// TwinCAT 3 PLC project Assembler
// ProgramVersion: 3.1.4023.0
// libraries:
//   Tc2_Standard, * (Beckhoff Automation GmbH)
//   Tc2_System, * (Beckhoff Automation GmbH)
//   Tc3_Module, * (Beckhoff Automation GmbH)
// project tree:
//   / GlobalTextList.TcGTLO, PlcTask.TcTTO, Visualization Manager.TcVMO (not stored)
//   POUs/ FB_Axxe.TcPOU, FB_Holder.TcPOU, FB_Nagel.TcPOU, FB_Robot.TcPOU, FB_Schraubendreher.TcPOU, MAIN.TcPOU, Mashine.TcPOU, Sensore.TcPOU
//   VISUs/ Visualization.TcVIS

CONFIGURATION Assembler
    RESOURCE PLC ON TwinCAT3
        TASK PlcTask(INTERVAL := T#10ms, PRIORITY := 20);
        PROGRAM MAIN WITH PlcTask : MAIN;
    END_RESOURCE
END_CONFIGURATION

// ---- POUs/MAIN.TcPOU
PROGRAM MAIN
VAR
	Position1:INT;
	Position2:INT;
	Position3:INT;
	MyMashine:Mashine;
END_VAR

MyMashine();

END_PROGRAM

// ---- POUs/Mashine.TcPOU
FUNCTION_BLOCK Mashine
VAR_INPUT
END_VAR
VAR_OUTPUT
END_VAR
VAR
	DelayTimer:TON;
	MyRobot:FB_Robot;
	l_Schraubendreher1:FB_Schraubendreher;
	l_Schraubendreher2:FB_Schraubendreher;
	l_i_Step_Stat:INT;
	l_i_Model1:INT:=0;
	l_i_Model2:INT:=0;
	l_i_Model3:INT:=0;
	l_i_Move_Step_Stat:INT;
	Holder:ARRAY[1..11] OF FB_Holder;
	Nagel:ARRAY[1..11] OF FB_Nagel;
	RoboCurrent:UINT:=1;
	Dre1Current:UINT:=1;
	Dre2Current:UINT:=1;
	DoneCurrent:uINT:=1;
	Sensore1:Sensore;
	Sensore2:Sensore;
	Sensore3:Sensore;
END_VAR

MyRobot.i_HOZAxxe.M_SetAxxeValues(AxxeMinPos:=0,AxxeMaxPos:=50);
MyRobot.i_GRFLeftAxxe.M_SetAxxeValues(AxxeMinPos:=0,AxxeMaxPos:=2);
MyRobot.i_GRFRightAxxe.M_SetAxxeValues(AxxeMinPos:=0,AxxeMaxPos:=-2);
l_Schraubendreher1.i_VTKAxxe.M_SetAxxeValues(AxxeMinPos:=0,AxxeMaxPos:=40);
l_Schraubendreher2.i_VTKAxxe.M_SetAxxeValues(AxxeMinPos:=0,AxxeMaxPos:=40);

//Move To Loading Position and Load Nail
IF NOT holder[RoboCurrent].Loaded AND RoboCurrent <= 11 THEN
	CASE l_i_Model1 OF
		0: 
			IF MoveToLoad(holder[RoboCurrent]) THEN
				l_i_Model1:=l_i_Model1+1;
			END_IF
		1:
			IF MyRobot.M_Load(holder[RoboCurrent])AND RoboCurrent < 11 THEN
				Nagel[RoboCurrent].visible:=TRUE;
				l_i_Model1:=l_i_Model1+1;
				RoboCurrent:=RoboCurrent+1;
			END_IF
		2:
			l_i_Model1:=0;
	END_CASE
END_IF
//if Loaded Move to Schraubendreher 1 and FestSchrauben
IF Holder[Dre1Current].Loaded THEN
	CASE l_i_Model2  OF
	0: 
	IF MoveToDreherOne(holder[Dre1Current]) THEN
		l_i_Model2:=l_i_Model2+1;	
	END_IF
	1:
	IF l_Schraubendreher1.M_Festschrauben(holder[Dre1Current]) AND Dre1Current < 11 THEN
		l_i_Model2:=l_i_Model2+1;
		Holder[Dre1Current].Loaded:=FALSE;
		Dre1Current:=Dre1Current+1;
	END_IF
	2:
	l_i_Model2:=0;
END_CASE
END_IF

//if it is Festgeschraubt then ab Schrauben
IF Holder[Dre2Current].Eingeschraubt THEN 
	CASE l_i_Model3 OF
	0: 
	IF MoveToDreherTwo(holder[Dre2Current]) THEN
		l_Schraubendreher2.Done:=FALSE;
		l_i_Model3:=l_i_Model3+1;
		
	END_IF
	1:
	IF l_Schraubendreher2.M_Abschrauben(holder[Dre2Current]) AND Dre2Current < 11 THEN
		l_i_Model3:=l_i_Model3+1;
		Dre2Current:=Dre2Current+1;
	END_IF
	2:
	l_i_Model3:=0;
END_CASE
END_IF


IF holder[DoneCurrent].Abgeschraubt THEN
	IF M_MoveOut(holder[DoneCurrent])  AND DoneCurrent < 11 THEN
		DoneCurrent:=DoneCurrent+1;
	END_IF
END_IF

METHOD Delay : BOOL
VAR_INPUT
END_VAR
DelayTimer(IN:=TRUE,PT:=T#500MS);
IF DelayTimer.Q THEN
	DelayTimer(IN:=FALSE);
	Delay:=TRUE;
END_IF
END_METHOD

METHOD M_MoveOut : BOOL
VAR_INPUT
	MyHolder : REFERENCE TO FB_Holder;
END_VAR
IF MyHolder.i_i_HolderPosition < 600 THEN
	MyHolder.MoveForward();
	MyHolder.Loaded:=FALSE;
	MyHolder.Eingeschraubt:=FALSE;
	Sensore3Active();
ELSE
	
	M_MoveOut:=TRUE;
END_IF
END_METHOD

METHOD MoveToDreherOne : BOOL
VAR_INPUT
	MyHolder: REFERENCE TO  FB_Holder;
END_VAR
IF NOT Sensore2Active() THEN
    MyHolder.MoveForward();
	 Sensore1Active();
ELSE
	MoveToDreherOne:=TRUE;
END_IF
END_METHOD

METHOD MoveToDreherTwo : BOOL
VAR_INPUT
	MyHolder: REFERENCE TO  FB_Holder;
END_VAR
IF NOT Sensore3Active() THEN
    MyHolder.MoveForward();
	 Sensore2Active();
ELSE
	MoveToDreherTwo:=TRUE;
END_IF
END_METHOD

METHOD MoveToLoad : BOOL
VAR_INPUT
	MyHolder: REFERENCE TO  FB_Holder;
END_VAR
IF NOT Sensore1Active() THEN
      MyHolder.MoveForward();
ELSE
	MoveToLoad:=TRUE;
END_IF
END_METHOD

METHOD Sensore1Active : BOOL
VAR_INPUT
END_VAR
IF Holder[RoboCurrent].i_i_HolderPosition = 85 THEN
	Sensore1.i_b_SensoreActive:=TRUE;
	Sensore1Active:=TRUE;
ELSE
	IF Holder[RoboCurrent].i_i_HolderPosition < 85 OR Holder[RoboCurrent].i_i_HolderPosition > 83 THEN
		Sensore1.i_b_SensoreActive:=FALSE;
		Sensore1Active:=FALSE;
	END_IF
END_IF
END_METHOD

METHOD Sensore2Active : BOOL
VAR_INPUT
END_VAR
IF Holder[Dre1Current].i_i_HolderPosition = 263 THEN
	Sensore2.i_b_SensoreActive:=TRUE;
	Sensore2Active:=TRUE;
ELSE
	IF Holder[Dre1Current].i_i_HolderPosition < 263 OR Holder[Dre1Current].i_i_HolderPosition > 263 THEN
		Sensore2.i_b_SensoreActive:=FALSE;
		Sensore2Active:=FALSE;
	END_IF
END_IF
END_METHOD

METHOD Sensore3Active : BOOL
VAR_INPUT
END_VAR
IF Holder[Dre2Current].i_i_HolderPosition = 404 THEN
	Sensore3.i_b_SensoreActive:=TRUE;
	Sensore3Active:=TRUE;
ELSE
	IF Holder[Dre2Current].i_i_HolderPosition < 404 OR Holder[Dre2Current].i_i_HolderPosition > 404 THEN
		Sensore3.i_b_SensoreActive:=FALSE;
		Sensore3Active:=FALSE;
	END_IF
END_IF
END_METHOD

END_FUNCTION_BLOCK

// ---- POUs/FB_Robot.TcPOU
FUNCTION_BLOCK FB_Robot
VAR_INPUT
	LoadDone:BOOL:=TRUE;
END_VAR
VAR_OUTPUT
END_VAR
VAR
	i_VTKAxxe:FB_Axxe;
	i_HOZAxxe:FB_Axxe;
	i_GRFLeftAxxe:FB_Axxe;
	i_GRFRightAxxe:FB_Axxe;
	l_i_Step_Stat:INT:=0;
	DelayTimer:TON;
	RoboNagel: FB_Nagel;
END_VAR

METHOD M_Delay : BOOL
VAR_INPUT
END_VAR
DelayTimer(IN:=TRUE,PT:=T#500ms);
IF DelayTimer.Q THEN
	DelayTimer(IN:=FALSE);
	M_Delay:=TRUE;
END_IF
END_METHOD

METHOD M_Load : BOOL
VAR_INPUT
	Myholder : REFERENCE TO FB_Holder; 
END_VAR
VAR
	
END_VAR
CASE l_i_Step_Stat OF
	0:
		IF M_RobotHOZLeft() THEN
			l_i_Step_Stat:=l_i_Step_Stat+1;
		END_IF
	1:
		
		IF i_VTKAxxe.M_SetAxxeValues(AxxeMinPos:=0,AxxeMaxPos:=25) THEN
			IF M_RobotVTKDown() THEN
				l_i_Step_Stat:=l_i_Step_Stat+1;
			END_IF
		END_IF
	2:
		LoadDone:=FALSE;
		IF M_RobotGRFZu() THEN
			l_i_Step_Stat:=l_i_Step_Stat+1;
			RoboNagel.visible:=true;
		END_IF
	3:
		IF M_RobotVTKUp() THEN
			l_i_Step_Stat:=l_i_Step_Stat+1;
		END_IF
	4:
		IF M_RobotHOZRight() THEN
				l_i_Step_Stat:=l_i_Step_Stat+1;	
		END_IF
	5:
		IF i_VTKAxxe.M_SetAxxeValues(AxxeMinPos:=0,AxxeMaxPos:=50) THEN
			IF M_RobotVTKDown() THEN
				l_i_Step_Stat:=l_i_Step_Stat+1;
				Myholder.Nagel.visible:=TRUE;
				RoboNagel.visible:=FALSE;
			END_IF
		END_IF
	6:
		IF M_RobotGRFAuf() THEN
			l_i_Step_Stat:=l_i_Step_Stat+1;
		END_IF
	7:	
		IF M_RobotVTKUp() THEN
			l_i_Step_Stat:=l_i_Step_Stat+1;
		END_IF
	8:	
		Myholder.Loaded:=true;
		LoadDone:=TRUE;
		M_Load:=TRUE;
		l_i_Step_Stat:=0;	
END_CASE
END_METHOD

METHOD M_RobotGRFAuf : BOOL
VAR_INPUT
END_VAR
IF i_GRFLeftAxxe.i_i_AxxePosition > i_GRFLeftAxxe.i_i_AxxeMinPos AND i_GRFRightAxxe.i_i_AxxePosition < i_GRFRightAxxe.i_i_AxxeMinPos THEN
	i_GRFLeftAxxe.i_i_AxxePosition := i_GRFLeftAxxe.i_i_AxxePosition-1;
	i_GRFRightAxxe.i_i_AxxePosition := i_GRFRightAxxe.i_i_AxxePosition+1;
	IF i_GRFLeftAxxe.i_i_AxxePosition = i_GRFLeftAxxe.i_i_AxxeMinPos AND i_GRFRightAxxe.i_i_AxxePosition = i_GRFRightAxxe.i_i_AxxeMinPos THEN
		IF M_Delay()THEN
			M_RobotGRFAuf:=TRUE;	
		END_IF
	END_IF
ELSE
	IF M_Delay()THEN
		M_RobotGRFAuf:=TRUE;	
	END_IF		
END_IF
END_METHOD

METHOD M_RobotGRFZu : BOOL
VAR_INPUT
END_VAR
IF i_GRFLeftAxxe.i_i_AxxePosition < i_GRFLeftAxxe.i_i_AxxeMaxPos AND i_GRFRightAxxe.i_i_AxxePosition > i_GRFRightAxxe.i_i_AxxeMaxPos THEN
	i_GRFLeftAxxe.i_i_AxxePosition := i_GRFLeftAxxe.i_i_AxxePosition+1;
	i_GRFRightAxxe.i_i_AxxePosition := i_GRFRightAxxe.i_i_AxxePosition-1;
	IF i_GRFLeftAxxe.i_i_AxxePosition = i_GRFLeftAxxe.i_i_AxxeMaxPos AND i_GRFRightAxxe.i_i_AxxePosition = i_GRFRightAxxe.i_i_AxxeMaxPos THEN
		IF M_Delay()THEN
			M_RobotGRFZu:=TRUE;	
		END_IF
	END_IF
ELSE
	IF M_Delay()THEN
		M_RobotGRFZu:=TRUE;	
	END_IF		
END_IF
END_METHOD

METHOD M_RobotHOZLeft : BOOL
VAR_INPUT
END_VAR
IF i_HOZAxxe.i_i_AxxePosition > i_VTKAxxe.i_i_AxxeMinPos THEN
i_HOZAxxe.i_i_AxxePosition := i_HOZAxxe.i_i_AxxePosition-1;
	IF i_HOZAxxe.i_i_AxxePosition = i_HOZAxxe.i_i_AxxeMinPos THEN
		IF M_Delay()THEN
			M_RobotHOZLeft:=TRUE;
		END_IF	
	END_IF
ELSE
	IF M_Delay()THEN
		M_RobotHOZLeft:=TRUE;	
	END_IF	
END_IF
END_METHOD

METHOD M_RobotHOZRight : BOOL
VAR_INPUT
END_VAR
IF i_HOZAxxe.i_i_AxxePosition < i_VTKAxxe.i_i_AxxeMaxPos THEN
i_HOZAxxe.i_i_AxxePosition := i_HOZAxxe.i_i_AxxePosition+1;
	IF i_HOZAxxe.i_i_AxxePosition = i_HOZAxxe.i_i_AxxeMaxPos THEN
		IF M_Delay()THEN
			M_RobotHOZRight:=TRUE;
		END_IF	
	END_IF
ELSE
	IF M_Delay()THEN
		M_RobotHOZRight:=TRUE;	
	END_IF	
END_IF
END_METHOD

METHOD M_RobotVTKDown : BOOL
VAR_INPUT
END_VAR
IF i_VTKAxxe.i_i_AxxePosition < i_VTKAxxe.i_i_AxxeMaxPos THEN
i_VTKAxxe.i_i_AxxePosition := i_VTKAxxe.i_i_AxxePosition+1;
	IF i_VTKAxxe.i_i_AxxePosition = i_VTKAxxe.i_i_AxxeMaxPos THEN
		IF M_Delay()THEN
			M_RobotVTKDown:=TRUE;
		END_IF	
	END_IF
ELSE
	IF M_Delay()THEN
		M_RobotVTKDown:=TRUE;	
	END_IF	
END_IF
END_METHOD

METHOD M_RobotVTKUp : BOOL
VAR_INPUT
END_VAR
IF i_VTKAxxe.i_i_AxxePosition > i_VTKAxxe.i_i_AxxeMinPos THEN
i_VTKAxxe.i_i_AxxePosition := i_VTKAxxe.i_i_AxxePosition-1;
	IF i_VTKAxxe.i_i_AxxePosition = i_VTKAxxe.i_i_AxxeMinPos THEN
		IF M_Delay()THEN
			M_RobotVTKUp:=TRUE;	
		END_IF	
	END_IF
ELSE
	IF M_Delay()THEN
		M_RobotVTKUp:=TRUE;	
	END_IF	
END_IF
END_METHOD

END_FUNCTION_BLOCK

// ---- POUs/FB_Axxe.TcPOU
FUNCTION_BLOCK FB_Axxe
VAR_INPUT
	i_i_AxxePosition	:	INT;
	i_i_AxxeMinPos		:	INT;
	i_i_AxxeMaxPos		:	INT;
END_VAR

METHOD M_SetAxxeValues : BOOL
VAR_INPUT
	AxxeMinPos		:	INT;
	AxxeMaxPos		:	INT;
END_VAR
i_i_AxxeMinPos:=AxxeMinPos;
i_i_AxxeMaxPos:=AxxeMaxPos;
IF i_i_AxxeMinPos = AxxeMinPos AND i_i_AxxeMaxPos = AxxeMaxPos THEN
	M_SetAxxeValues:=TRUE;	
END_IF
END_METHOD

END_FUNCTION_BLOCK

// ---- POUs/FB_Nagel.TcPOU
FUNCTION_BLOCK FB_Nagel
VAR_INPUT
	visible:BOOL;
END_VAR

END_FUNCTION_BLOCK

// ---- POUs/FB_Holder.TcPOU
FUNCTION_BLOCK FB_Holder
VAR_INPUT
	i_i_HolderPosition:	INT;
	Loaded:BOOL;
	Eingeschraubt	:	BOOL;
	Abgeschraubt: BOOL;
	Nagel: FB_Nagel;
END_VAR

METHOD MoveForward : BOOL
VAR_INPUT

END_VAR
i_i_HolderPosition:=i_i_HolderPosition+1;
END_METHOD

END_FUNCTION_BLOCK

// ---- POUs/FB_Schraubendreher.TcPOU
FUNCTION_BLOCK FB_Schraubendreher
VAR_INPUT
	Done:BOOL:=TRUE;
END_VAR
VAR
	i_VTKAxxe:FB_Axxe;
	l_b_Power:BOOL;
	l_i_Step_Stat:INT;
	DelayTimer:TON;
END_VAR

METHOD M_Abschrauben : BOOL
VAR_INPUT
	MyHolder:REFERENCE TO FB_Holder;
END_VAR
CASE l_i_Step_Stat OF
	0: 
		IF M_Turn() THEN
			l_i_Step_Stat:=l_i_Step_Stat+1;	
		END_IF
	1:		
		IF M_SchraubendreherDown() THEN
			l_i_Step_Stat:=l_i_Step_Stat+1;
		END_IF
	2:
		IF M_SchraubendreherUp() THEN
			l_i_Step_Stat:=l_i_Step_Stat+1;
		END_IF
	3: 
		IF M_Turn() THEN
			l_i_Step_Stat:=0;
			done:=TRUE;
			MyHolder.Eingeschraubt:=FALSE;
			MyHolder.Abgeschraubt:=TRUE;
			M_Abschrauben:=true;	
		END_IF
END_CASE
END_METHOD

METHOD M_Delay : BOOL
VAR_INPUT
END_VAR
DelayTimer(IN:=TRUE,PT:=T#500ms);
IF DelayTimer.Q THEN
	DelayTimer(IN:=FALSE);
	M_Delay:=TRUE;
END_IF
END_METHOD

METHOD M_Festschrauben : BOOL
VAR_INPUT
	MyHolder:REFERENCE TO FB_Holder;
END_VAR
CASE l_i_Step_Stat OF
	0: 
		IF M_Turn() THEN
			l_i_Step_Stat:=l_i_Step_Stat+1;
		END_IF
	1:		
		IF M_SchraubendreherDown() THEN
			l_i_Step_Stat:=l_i_Step_Stat+1;
		END_IF
	2:
		IF M_SchraubendreherUp() THEN
			l_i_Step_Stat:=l_i_Step_Stat+1;
		END_IF
	3: 
		IF M_Turn() THEN
			l_i_Step_Stat:=0;
			done:=TRUE;
			MyHolder.Eingeschraubt:=TRUE;
			M_Festschrauben:=TRUE;	
		END_IF
END_CASE
END_METHOD

METHOD M_SchraubendreherDown : BOOL
VAR_INPUT
END_VAR
IF i_VTKAxxe.i_i_AxxePosition < i_VTKAxxe.i_i_AxxeMaxPos THEN
i_VTKAxxe.i_i_AxxePosition := i_VTKAxxe.i_i_AxxePosition+1;
	IF i_VTKAxxe.i_i_AxxePosition = i_VTKAxxe.i_i_AxxeMaxPos THEN
		IF M_Delay()THEN
			M_SchraubendreherDown:=TRUE;
		END_IF	
	END_IF
ELSE
	IF M_Delay()THEN
		M_SchraubendreherDown:=TRUE;	
	END_IF	
END_IF
END_METHOD

METHOD M_SchraubendreherUp : BOOL
VAR_INPUT
END_VAR
IF i_VTKAxxe.i_i_AxxePosition > i_VTKAxxe.i_i_AxxeMinPos THEN
i_VTKAxxe.i_i_AxxePosition := i_VTKAxxe.i_i_AxxePosition-1;
	IF i_VTKAxxe.i_i_AxxePosition = i_VTKAxxe.i_i_AxxeMinPos THEN
		IF M_Delay()THEN
			M_SchraubendreherUp:=TRUE;	
		END_IF	
	END_IF
ELSE
	IF M_Delay()THEN
		M_SchraubendreherUp:=TRUE;	
	END_IF	
END_IF
END_METHOD

METHOD M_Turn : BOOL
VAR_INPUT
END_VAR
l_b_Power:=NOT l_b_Power;
M_Turn:=TRUE;
END_METHOD

END_FUNCTION_BLOCK

// ---- POUs/Sensore.TcPOU
FUNCTION_BLOCK Sensore
VAR_INPUT
	i_i_SensorePosition	:	INT;
	i_b_SensoreActive		:	BOOL;
END_VAR

END_FUNCTION_BLOCK

// ---- VISUs/Visualization.TcVIS
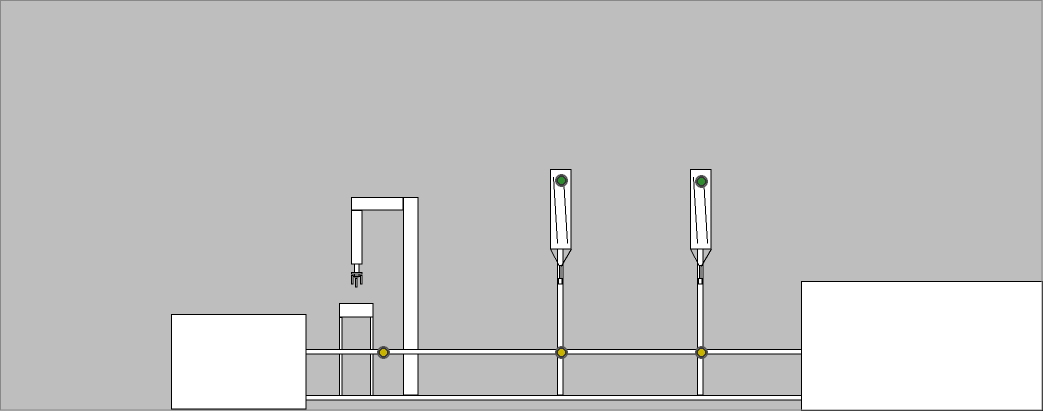
VISUALIZATION Visualization  // 1043x411
    Group (352,275 8x12), invisible if: NOT MAIN.MyMashine.MyRobot.RoboNagel.visible
        p3560616238: MAIN.MyMashine.MyRobot.i_HOZAxxe.i_i_AxxePosition
        p2738717112: MAIN.MyMashine.MyRobot.i_VTKAxxe.i_i_AxxePosition
        Ellipse (0,0 8x2)
        Rectangle (3,3 2x9)
    Rectangle (370,316 3x84)
    Rectangle (339,317 3x83)
    Rectangle (403,197 15x198)
    Rectangle (697,197 6x198)
    Rectangle (557,197 6x198)
    Rectangle (261,349 636x5)
    Rectangle (259,395 637x5)
    Ellipse (242,348 48x54)
    Group (293,327 8x12), invisible if: NOT MAIN.MyMashine.Holder[1].Nagel.visible
        p3560616238: MAIN.MyMashine.Holder[1].i_i_HolderPosition
        Ellipse (0,0 8x2)
        Rectangle (3,3 2x9)
    RoundedRectangle (290,339 13x10)
        p3560616238: MAIN.MyMashine.Holder[1].i_i_HolderPosition
    RoundedRectangle (290,339 13x10)
        p3560616238: MAIN.MyMashine.Holder[4].i_i_HolderPosition
    Group (293,327 8x12), invisible if: NOT MAIN.MyMashine.Holder[4].Nagel.visible
        p3560616238: MAIN.MyMashine.Holder[4].i_i_HolderPosition
        Ellipse (0,0 8x2)
        Rectangle (3,3 2x9)
    RoundedRectangle (290,339 13x10)
        p3560616238: MAIN.MyMashine.Holder[3].i_i_HolderPosition
    Group (293,327 8x12), invisible if: NOT MAIN.MyMashine.Holder[3].Nagel.visible
        p3560616238: MAIN.MyMashine.Holder[3].i_i_HolderPosition
        Ellipse (0,0 8x2)
        Rectangle (3,3 2x9)
    RoundedRectangle (290,339 13x10)
        p3560616238: MAIN.MyMashine.Holder[2].i_i_HolderPosition
    Group (293,327 8x12), invisible if: NOT MAIN.MyMashine.Holder[2].Nagel.visible
        p3560616238: MAIN.MyMashine.Holder[2].i_i_HolderPosition
        Ellipse (0,0 8x2)
        Rectangle (3,3 2x9)
    Rectangle (351,197 52x13)
    Group (351,210 11x74)
        p3560616238: MAIN.MyMashine.MyRobot.i_HOZAxxe.i_i_AxxePosition
        Rectangle (9,65 2x9)
            p3560616238: MAIN.MyMashine.MyRobot.i_GRFRightAxxe.i_i_AxxePosition
            p2738717112: MAIN.MyMashine.MyRobot.i_VTKAxxe.i_i_AxxePosition
        Rectangle (0,65 2x9)
            p3560616238: MAIN.MyMashine.MyRobot.i_GRFLeftAxxe.i_i_AxxePosition
            p2738717112: MAIN.MyMashine.MyRobot.i_VTKAxxe.i_i_AxxePosition
        Rectangle (3,1 5x65)
            p2738717112: MAIN.MyMashine.MyRobot.i_VTKAxxe.i_i_AxxePosition
        Rectangle (0,62 11x2)
            p2738717112: MAIN.MyMashine.MyRobot.i_VTKAxxe.i_i_AxxePosition
        Rectangle (0,0 11x54)
    Group (550,169 21x115)
        p2738717112: MAIN.MyMashine.l_Schraubendreher1.i_VTKAxxe.i_i_AxxePosition
        Rectangle (0,0 21x80)
        Line (21,80) (11,97)
        Line (0,80) (9,97)
        RoundedRectangle (9,96 2x14)
        Rectangle (8,109 4x6)
        Line (13,8) (17,74)
        Line (3,8) (7,74)
        Lamp1 (4,4 15x15), variable: MAIN.MyMashine.l_Schraubendreher1.l_b_Power, style: Lamp-Lamp1-Green
    Group (690,169 21x115)
        p2738717112: MAIN.MyMashine.l_Schraubendreher2.i_VTKAxxe.i_i_AxxePosition
        Rectangle (0,0 21x80)
        Line (21,80) (11,97)
        Line (0,80) (9,97)
        RoundedRectangle (9,96 2x14)
        Rectangle (8,109 4x6)
        Line (13,8) (17,74)
        Line (3,8) (7,74)
        Lamp1 (4,5 15x15), variable: MAIN.MyMashine.l_Schraubendreher2.l_b_Power, style: Lamp-Lamp1-Green
    Lamp1 (554,345 15x15), variable: MAIN.MyMashine.Sensore2.i_b_SensoreActive, style: Lamp-Lamp1-Yellow
    Lamp1 (694,345 15x15), variable: MAIN.MyMashine.Sensore3.i_b_SensoreActive, style: Lamp-Lamp1-Yellow
    Rectangle (339,303 34x14)
    RoundedRectangle (290,338 13x10)
        p3560616238: MAIN.MyMashine.Holder[11].i_i_HolderPosition
    Group (293,326 8x12), invisible if: NOT MAIN.MyMashine.Holder[2].Nagel.visible
        p3560616238: MAIN.MyMashine.Holder[11].i_i_HolderPosition
        Ellipse (0,0 8x2)
        Rectangle (3,3 2x9)
    RoundedRectangle (290,339 13x10)
        p3560616238: MAIN.MyMashine.Holder[9].i_i_HolderPosition
    Group (293,327 8x12), invisible if: NOT MAIN.MyMashine.Holder[2].Nagel.visible
        p3560616238: MAIN.MyMashine.Holder[9].i_i_HolderPosition
        Ellipse (0,0 8x2)
        Rectangle (3,3 2x9)
    RoundedRectangle (291,339 13x10)
        p3560616238: MAIN.MyMashine.Holder[8].i_i_HolderPosition
    Group (294,325 8x12), invisible if: NOT MAIN.MyMashine.Holder[8].Nagel.visible
        p3560616238: MAIN.MyMashine.Holder[8].i_i_HolderPosition
        Ellipse (0,0 8x2)
        Rectangle (3,3 2x9)
    RoundedRectangle (290,339 13x10)
        p3560616238: MAIN.MyMashine.Holder[7].i_i_HolderPosition
    Group (293,327 8x12), invisible if: NOT MAIN.MyMashine.Holder[7].Nagel.visible
        p3560616238: MAIN.MyMashine.Holder[7].i_i_HolderPosition
        Ellipse (0,0 8x2)
        Rectangle (3,3 2x9)
    RoundedRectangle (291,339 13x10)
        p3560616238: MAIN.MyMashine.Holder[6].i_i_HolderPosition
    Group (294,327 8x12), invisible if: NOT MAIN.MyMashine.Holder[6].Nagel.visible
        p3560616238: MAIN.MyMashine.Holder[6].i_i_HolderPosition
        Ellipse (0,0 8x2)
        Rectangle (3,3 2x9)
    RoundedRectangle (290,339 13x10)
        p3560616238: MAIN.MyMashine.Holder[5].i_i_HolderPosition
    Group (293,326 8x12), invisible if: NOT MAIN.MyMashine.Holder[5].Nagel.visible
        p3560616238: MAIN.MyMashine.Holder[5].i_i_HolderPosition
        Ellipse (0,0 8x2)
        Rectangle (3,3 2x9)
    Lamp1 (376,345 15x15), variable: MAIN.MyMashine.Sensore1.i_b_SensoreActive, style: Lamp-Lamp1-Yellow
    Rectangle (801,281 242x130)
    Rectangle (171,314 135x95)
END_VISUALIZATION
